(* CODESYS project CAN_MIR3502.20200326.1.project
   Description: Receives some incoming messages and echoes them with CAN-ID +1
   Title: CAN Bus API Example
   Version: 1.0.0.0
   Company: 3S - Smart Software Solutions GmbH
   Author: 3S - Smart Software Solutions GmbH

Project tree, tasks and I/O mapping:
  Device : Changsha-Cyber-MI-linux, Changsha Cyber-MI Co., Ltd., version 3.5.10.40
    application Application
      libraries: CAN API, 1.0.0.3 (3S - Smart Software Solutions GmbH); Standard, * (System)
      task MainTask (cyclic, interval t#20ms, priority 1) calls prg_mir3502
      function blocks/
        function block MsgProcessorMIR3502 [ST]: ProcessMessage
        function block FB_MIR3502_CAN [ST]: setup_sendmsg
        function block fb_avg [ST]
      global variables GVL
      program prg_mir3502 [ST]
      trace Trace (task MainTask): prg_mir3502.ai_00
    SoftMotion General Axis Pool
*)

// Device/Application/GVL
VAR_GLOBAL

END_VAR

// Device/Application/prg_mir3502
PROGRAM prg_mir3502
VAR
	// CAN 0 ,  250K bps,  buffer size: 100
	CanConfig	: CAN.DRIVER_CONFIG := (usiNetwork:= 0, uiBaudrate:= 250, ctMessages:= 100);
	CANdriver	: CAN.CANBus_29bit :=  (DriverConfig:= CanConfig);
	
	// MIR3502
	MIR3502 : FB_MIR3502_CAN := (xEnable := TRUE);
	avg_ai00:fb_avg := (num := 32);
	
	ai_00_raw:DINT;
	ai_00 : DINT;
	ai_06 : DINT;
	ai_12 : DINT;
END_VAR


/// Run  the CAN Driver
CANdriver(DriverConfig:= CanConfig, eError=> );

MIR3502(CANdriver := CANdriver);

//设置扩展IO模块的DO， PWM
MIR3502.xDO[3] := TRUE;
MIR3502.xDO[12] := TRUE;

//设置哪些AI需要读取，没有设置的AI值不会送到主控制器，以降低CAN总线负载率
MIR3502.xEnable_AI[00] := TRUE;
MIR3502.xEnable_AI[06] := TRUE;
MIR3502.xEnable_AI[12] := TRUE;

//读取扩展IO模块的AI
ai_00_raw := MIR3502.uiAI[0];
avg_ai00(in_val := ai_00_raw, out_val => ai_00);
ai_06 := MIR3502.uiAI[6];
ai_12 := MIR3502.uiAI[12];

END_PROGRAM

// Device/Application/function blocks/FB_MIR3502_CAN
FUNCTION_BLOCK FB_MIR3502_CAN
VAR_INPUT
	xEnable:BOOL := FALSE;
	xEnable_AI:ARRAY[0..31] OF BOOL := [32(FALSE)];
	xDO:ARRAY[0..23] OF BOOL := [24(FALSE)];
	uiPWM:ARRAY[0..1] OF UINT := [2(0)];
END_VAR
VAR_IN_OUT
	CANdriver	: CAN.CANBus_29bit;
END_VAR
VAR_OUTPUT
	uiAI:ARRAY[0..31] OF UINT;
    xDI:ARRAY[0..31] OF BOOL;
    Vcc:UINT;
    xError:BOOL := FALSE;
    sError:STRING(128) := 'No Error';	
	uiStat : UINT := 0;
END_VAR
VAR
	stat:UINT := 0;
	i :UINT := 0;
	recver:can.RECEIVER_AREA;
	areaReceiver:CAN.CANAreaReceiver;
	msgProcessor:MsgProcessorMIR3502;
	hAreaReceiver	: CAN.CAA.HANDLE := CAN.CAA.gc_hINVALID;
	bData:BYTE;
	msg_send :CAN.MESSAGE;
	msg_recv :CAN.MESSAGE;
END_VAR


CASE stat OF
0:
	FOR i := 0 TO 31 DO
		xEnable_AI[i] := FALSE;
		uiAI[i] := 0;
	END_FOR	
	
	FOR i := 0 TO 23 DO
		xDO[i] := FALSE;
		xDI[i] := FALSE;
	END_FOR
	
	FOR i := 0 TO 1 DO
		uiPWM[i] := 0;
	END_FOR
	
	Vcc := 0;
	xError := FALSE;
	sError := 'No Error';
	
	recver.dwIdStart := 300;
	recver.dwIdEnd := 308;
	recver.xRTRMask := FALSE;
	recver.xRTRValue := FALSE;
	recver.xTransmitMask := FALSE;
	recver.xTransmitValue := FALSE;

	hAreaReceiver := CANdriver.GetAreaReceiver(recver, eError=>);

	stat := 10;
	
10:  //wait enable
	IF xEnable THEN
		stat := 20;
	END_IF

20: //send
	setup_sendmsg();
	CANdriver.SendMessage(msg_send, eError=>);
	stat := 30;

30: //wait for receive
	stat := 20;  //send next msg
	
END_CASE

uiStat := stat;

CANdriver.ReceiveMessage(hReceiver := hAreaReceiver, itfMsgProcessor := msgProcessor, tTimeLimit := T#5MS, eError=>);

msgProcessor(CANdriver := CANdriver);

FOR i := 0 TO 31 DO
	uiAI[i] := msgProcessor.uiAI[i];
	xDI[i] := msgProcessor.xDI[i];
	Vcc := msgProcessor.Vcc;
END_FOR

ACTION setup_sendmsg:
	bData.0 := xDO[0]; 
	bData.1 := xDO[1];
	bData.2 := xDO[2];
	bData.3 := xDO[3];
	bData.4 := xDO[4];
	bData.5 := xDO[5];
	bData.6 := xDO[6];
	bData.7 := xDO[7];
	msg_send.abyData[0] := bData;
	
	bData.0 := xDO[8]; 
	bData.1 := xDO[9];
	bData.2 := xDO[10];
	bData.3 := xDO[11];
	bData.4 := xDO[12];
	bData.5 := xDO[13];
	bData.6 := xDO[14];
	bData.7 := xDO[15];
	msg_send.abyData[1] := bData;	
	
	bData.0 := xDO[16]; 
	bData.1 := xDO[17];
	bData.2 := xDO[18];
	bData.3 := xDO[19];
	bData.4 := xDO[20];
	bData.5 := xDO[21];
	bData.6 := xDO[22];
	bData.7 := xDO[23];
	msg_send.abyData[2] := bData;	

	bData.0 := NOT (xEnable_AI[0] OR xEnable_AI[1] OR xEnable_AI[2] OR xEnable_AI[3]) ; 
	bData.1 := NOT (xEnable_AI[4] OR xEnable_AI[5] OR xEnable_AI[6] OR xEnable_AI[7]) ; 
	bData.2 := NOT (xEnable_AI[8] OR xEnable_AI[9] OR xEnable_AI[10] OR xEnable_AI[11]) ; 
	bData.3 := NOT (xEnable_AI[12] OR xEnable_AI[13] OR xEnable_AI[14] OR xEnable_AI[15]) ; 
	bData.4 := NOT (xEnable_AI[16] OR xEnable_AI[17] OR xEnable_AI[18] OR xEnable_AI[19]) ; 
	bData.5 := NOT (xEnable_AI[20] OR xEnable_AI[21] OR xEnable_AI[22] OR xEnable_AI[23]) ; 
	bData.6 := NOT (xEnable_AI[24] OR xEnable_AI[25] OR xEnable_AI[26] OR xEnable_AI[27]) ; 
	bData.7 := NOT (xEnable_AI[28] OR xEnable_AI[29] OR xEnable_AI[30] OR xEnable_AI[31]) ; 
	msg_send.abyData[3] := bData;	
	
	bData := ANY_TO_BYTE(uiPWM[0] MOD 256);
	msg_send.abyData[4] := bData;
	
	bData := ANY_TO_BYTE(uiPWM[0] / 256);
	msg_send.abyData[5] := bData;
	
	bData := ANY_TO_BYTE(uiPWM[1] MOD 256);
	msg_send.abyData[6] := bData;
	
	bData := ANY_TO_BYTE(uiPWM[1] / 256);
	msg_send.abyData[7] := bData;
	
	msg_send.udiCanID := 400;
	msg_send.usiDataLength := 8;
	msg_send.xIs29BitMessage := FALSE;
	msg_send.xRTR := FALSE;
END_ACTION

END_FUNCTION_BLOCK

// Device/Application/function blocks/MsgProcessorMIR3502
FUNCTION_BLOCK MsgProcessorMIR3502 IMPLEMENTS CAN.IMessageProcessor
VAR_IN_OUT
	CANdriver	: CAN.CANBus_29bit;
END_VAR
VAR_OUTPUT
	uiAI:ARRAY[0..31] OF UINT;
    xDI:ARRAY[0..31] OF BOOL;
    Vcc:UINT;	
END_VAR
VAR
	_pCANdriver : POINTER TO CAN.CANBus_29bit;
END_VAR

_pCANdriver := ADR(CANdriver);

METHOD ProcessMessage
VAR_IN_OUT
	(* The messages received by the receiver *)
	Message	: CAN.RxMessage;
END_VAR

VAR
	id:UDINT;
END_VAR
IF _pCANdriver = 0 THEN
	RETURN;
END_IF

id := Message.udiCanID;

CASE id OF 
300:  //ai-00  ~  ai-03
	uiAI[0] := ANY_TO_UINT(Message.abyData[1])*256 + Message.abyData[0];
	uiAI[1] := ANY_TO_UINT(Message.abyData[3])*256 + Message.abyData[2];
	uiAI[2] := ANY_TO_UINT(Message.abyData[5])*256 + Message.abyData[4];
	uiAI[3] := ANY_TO_UINT(Message.abyData[7])*256 + Message.abyData[6];
 301:
	uiAI[4] := ANY_TO_UINT(Message.abyData[1])*256 + Message.abyData[0];
	uiAI[5] := ANY_TO_UINT(Message.abyData[3])*256 + Message.abyData[2];
	uiAI[6] := ANY_TO_UINT(Message.abyData[5])*256 + Message.abyData[4];
	uiAI[7] := ANY_TO_UINT(Message.abyData[7])*256 + Message.abyData[6];
 302:
	uiAI[8] := ANY_TO_UINT(Message.abyData[1])*256 + Message.abyData[0];
	uiAI[9] := ANY_TO_UINT(Message.abyData[3])*256 + Message.abyData[2];
	uiAI[10] := ANY_TO_UINT(Message.abyData[5])*256 + Message.abyData[4];
	uiAI[11] := ANY_TO_UINT(Message.abyData[7])*256 + Message.abyData[6];
 303:
	uiAI[12] := ANY_TO_UINT(Message.abyData[1])*256 + Message.abyData[0];
	uiAI[13] := ANY_TO_UINT(Message.abyData[3])*256 + Message.abyData[2];
	uiAI[14] := ANY_TO_UINT(Message.abyData[5])*256 + Message.abyData[4];
	uiAI[15] := ANY_TO_UINT(Message.abyData[7])*256 + Message.abyData[6];
 304:
	uiAI[16] := ANY_TO_UINT(Message.abyData[1])*256 + Message.abyData[0];
	uiAI[17] := ANY_TO_UINT(Message.abyData[3])*256 + Message.abyData[2];
	uiAI[18] := ANY_TO_UINT(Message.abyData[5])*256 + Message.abyData[4];
	uiAI[19] := ANY_TO_UINT(Message.abyData[7])*256 + Message.abyData[6];
 305:
	uiAI[20] := ANY_TO_UINT(Message.abyData[1])*256 + Message.abyData[0];
	uiAI[21] := ANY_TO_UINT(Message.abyData[3])*256 + Message.abyData[2];
	uiAI[22] := ANY_TO_UINT(Message.abyData[5])*256 + Message.abyData[4];
	uiAI[23] := ANY_TO_UINT(Message.abyData[7])*256 + Message.abyData[6];
 306:
	uiAI[24] := ANY_TO_UINT(Message.abyData[1])*256 + Message.abyData[0];
	uiAI[25] := ANY_TO_UINT(Message.abyData[3])*256 + Message.abyData[2];
	uiAI[26] := ANY_TO_UINT(Message.abyData[5])*256 + Message.abyData[4];
	uiAI[27] := ANY_TO_UINT(Message.abyData[7])*256 + Message.abyData[6];
 307:
	uiAI[28] := ANY_TO_UINT(Message.abyData[1])*256 + Message.abyData[0];
	uiAI[29] := ANY_TO_UINT(Message.abyData[3])*256 + Message.abyData[2];
	uiAI[30] := ANY_TO_UINT(Message.abyData[5])*256 + Message.abyData[4];
	uiAI[31] := ANY_TO_UINT(Message.abyData[7])*256 + Message.abyData[6];
 308:  //DI00 ~ DI23   and  Vcc
	xDi[0] :=  Message.abyData[0].0;
	xDi[1] :=  Message.abyData[0].1;
	xDi[2] :=  Message.abyData[0].2;
	xDi[3] :=  Message.abyData[0].3;
	xDi[4] :=  Message.abyData[0].4;
	xDi[5] :=  Message.abyData[0].5;
	xDi[6] :=  Message.abyData[0].6;
	xDi[7] :=  Message.abyData[0].7;
	
	xDi[8] :=  Message.abyData[1].0;
	xDi[9] :=  Message.abyData[1].1;
	xDi[10] :=  Message.abyData[1].2;
	xDi[11] :=  Message.abyData[1].3;
	xDi[12] :=  Message.abyData[1].4;
	xDi[13] :=  Message.abyData[1].5;
	xDi[14] :=  Message.abyData[1].6;
	xDi[15] :=  Message.abyData[1].7;

	xDi[16] :=  Message.abyData[2].0;
	xDi[17] :=  Message.abyData[2].1;
	xDi[18] :=  Message.abyData[2].2;
	xDi[19] :=  Message.abyData[2].3;
	xDi[20] :=  Message.abyData[2].4;
	xDi[21] :=  Message.abyData[2].5;
	xDi[22] :=  Message.abyData[2].6;
	xDi[23] :=  Message.abyData[2].7;

	xDi[24] :=  Message.abyData[3].0;
	xDi[25] :=  Message.abyData[3].1;
	xDi[26] :=  Message.abyData[3].2;
	xDi[27] :=  Message.abyData[3].3;
	xDi[28] :=  Message.abyData[3].4;
	xDi[29] :=  Message.abyData[3].5;
	xDi[30] :=  Message.abyData[3].6;
	xDi[31] :=  Message.abyData[3].7;	
	
	Vcc := ANY_TO_UINT(Message.abyData[7])*256 + Message.abyData[6];
END_CASE
END_METHOD

END_FUNCTION_BLOCK

// Device/Application/function blocks/fb_avg
FUNCTION_BLOCK fb_avg
VAR_INPUT
	in_val:DINT;
	num:DINT := 10;
END_VAR
VAR_OUTPUT
	out_val:DINT;
END_VAR
VAR
	num_max : DINT := 255;
	data:ARRAY[1..255] OF DINT; //需要与上面的num_max保持一致
	ptr :UINT := 1;
	i: DINT;
	sum: DINT;
END_VAR

IF num <1 THEN
	out_val := 0;
	RETURN;
END_IF
IF num > num_max THEN
	num := num_max;
END_IF

data[ptr] := in_val;
ptr := ptr + 1;
IF ptr > num THEN
	ptr := 1;
END_IF

sum := 0;
FOR i := 1 TO num DO
	sum := sum + data[i];
END_FOR

out_val := sum/num;

END_FUNCTION_BLOCK
